TYPE ST_IOOutput :
STRUCT
	QxLampeRouge AT%Q*:BOOL;
	QxLampeVerte AT%Q* : BOOL;
	QxLampeOrange AT%Q* :BOOL;
END_STRUCT
END_TYPE

(* stored: Version 1.1.0.1, ProductVersion 3.1.4020.6
   DUT ST_IOOutput: Id {eb339f95-e975-4425-8e88-c959e46d7639} *)
